{attribute 'qualified_only'}
VAR_GLOBAL
	stanprzycisku:BOOL;
END_VAR

(* stored: Version 1.1.0.1, ProductVersion 3.1.4024.4
   GVL DVL: Id {1459322e-ca6a-4d1e-b275-1a3a645bf410} *)
